// TIA Portal V17 export
// export: Created 2025-03-05T08:00:04.2235864Z, ExportSetting WithDefaults, DisplayName Totally Integrated Automation Portal, DisplayVersion V17 Update 8, DisplayName TIA Portal Openness, DisplayVersion V17 Update 8, DisplayName TIA Portal Version Control Interface, DisplayVersion V17, DisplayName SINAMICS Startdrive Advanced, DisplayVersion V17 SP2, DisplayName SINAMICS Startdrive G110M, G120, G120C, G120D, G120P, G115D, DisplayVersion V17 SP2, DisplayName SINAMICS Startdrive G130, G150, S120, S150, SINAMICS MV, S210, DisplayVersion V17 SP2, DisplayName STEP 7 Professional, DisplayVersion V17 Update 8, DisplayName SINUMERIK ONE STEP 7 Toolbox, DisplayVersion V17 Update 12, DisplayName SINUMERIK 840D sl STEP 7 Toolbox, DisplayVersion V17 Update 12, DisplayName STEP 7 Safety, DisplayVersion V17 Update 6, DisplayName WinCC Advanced, DisplayVersion V17 Update 8
FUNCTION "FC2037_GANTRY_ROBOT_TEST_CYCLE" : Void   // FC2037, LAD
{ S7_Optimized_Access := 'FALSE' }
AUTHOR : ETXETAR
VERSION : 1.0
// stored: AutoNumber false, IsIECCheckEnabled false, SetENOAutomatically false, UDAEnableTagReadback false
   VAR CONSTANT
      FC_NUMBER : DInt := 2037;
   END_VAR
   VAR_TEMP   // added for the SCL form of the ladder/FBD networks
      _w1 : Bool;
      _w2 : Bool;
   END_VAR
BEGIN

REGION Network 1: CHANGE CYCLE GENERAL CONDITIONS
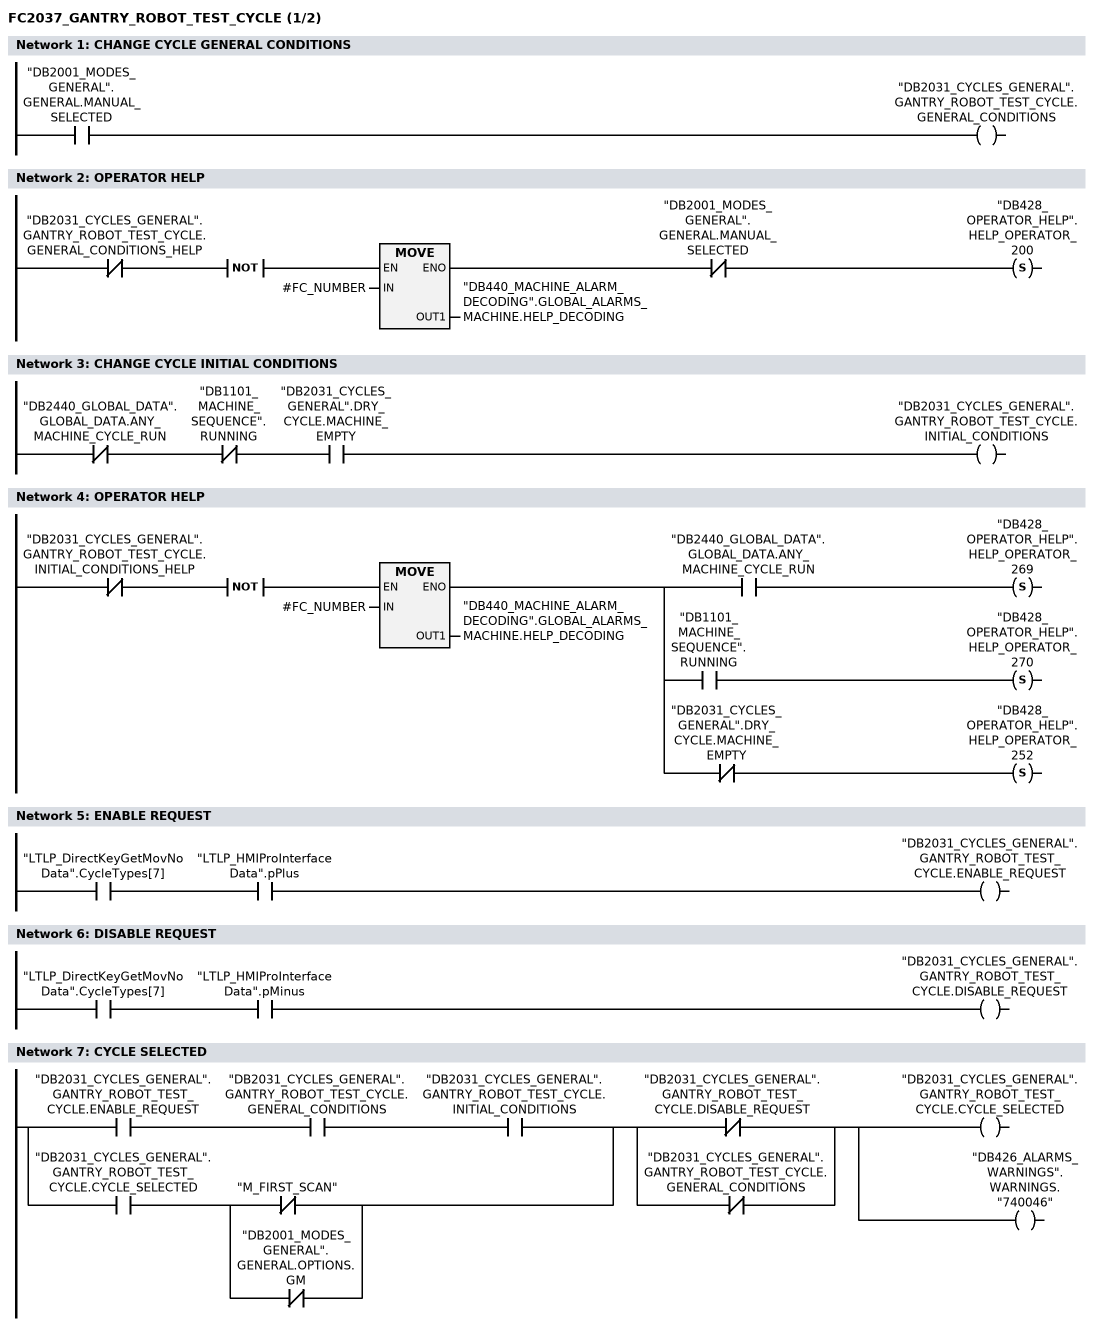
   RUNG wire#powerrail
      Contact( "DB2001_MODES_GENERAL".GENERAL.MANUAL_SELECTED )
      Coil( "DB2031_CYCLES_GENERAL".GANTRY_ROBOT_TEST_CYCLE.GENERAL_CONDITIONS )
   END_RUNG
   // the same network as SCL:
   "DB2031_CYCLES_GENERAL".GANTRY_ROBOT_TEST_CYCLE.GENERAL_CONDITIONS := "DB2001_MODES_GENERAL".GENERAL.MANUAL_SELECTED;
END_REGION

REGION Network 2: OPERATOR HELP
   RUNG wire#powerrail
      I_Contact( "DB2031_CYCLES_GENERAL".GANTRY_ROBOT_TEST_CYCLE.GENERAL_CONDITIONS_HELP )
      Not()
      { S7_GenerateENO := "TRUE" } Move(in := #FC_NUMBER, out1 => "DB440_MACHINE_ALARM_DECODING".GLOBAL_ALARMS_MACHINE.HELP_DECODING)
      I_Contact( "DB2001_MODES_GENERAL".GENERAL.MANUAL_SELECTED )
      S_Coil( "DB428_OPERATOR_HELP".HELP_OPERATOR_200 )
   END_RUNG
   // the same network as SCL:
   // ENO of a box is taken as its EN; it also drops when the box reports an error
   #_w1 := NOT (NOT "DB2031_CYCLES_GENERAL".GANTRY_ROBOT_TEST_CYCLE.GENERAL_CONDITIONS_HELP);
   IF #_w1 THEN "DB440_MACHINE_ALARM_DECODING".GLOBAL_ALARMS_MACHINE.HELP_DECODING := #FC_NUMBER; END_IF;
   IF #_w1 AND NOT "DB2001_MODES_GENERAL".GENERAL.MANUAL_SELECTED THEN
       "DB428_OPERATOR_HELP".HELP_OPERATOR_200 := TRUE;
   END_IF;
END_REGION

REGION Network 3: CHANGE CYCLE INITIAL CONDITIONS
   RUNG wire#powerrail
      I_Contact( "DB2440_GLOBAL_DATA".GLOBAL_DATA.ANY_MACHINE_CYCLE_RUN )
      I_Contact( "DB1101_MACHINE_SEQUENCE".RUNNING )
      Contact( "DB2031_CYCLES_GENERAL".DRY_CYCLE.MACHINE_EMPTY )
      Coil( "DB2031_CYCLES_GENERAL".GANTRY_ROBOT_TEST_CYCLE.INITIAL_CONDITIONS )
   END_RUNG
   // the same network as SCL:
   "DB2031_CYCLES_GENERAL".GANTRY_ROBOT_TEST_CYCLE.INITIAL_CONDITIONS := NOT "DB2440_GLOBAL_DATA".GLOBAL_DATA.ANY_MACHINE_CYCLE_RUN AND NOT "DB1101_MACHINE_SEQUENCE".RUNNING AND "DB2031_CYCLES_GENERAL".DRY_CYCLE.MACHINE_EMPTY;
END_REGION

REGION Network 4: OPERATOR HELP
   RUNG wire#powerrail
      I_Contact( "DB2031_CYCLES_GENERAL".GANTRY_ROBOT_TEST_CYCLE.INITIAL_CONDITIONS_HELP )
      Not()
      { S7_GenerateENO := "TRUE" } Move(in := #FC_NUMBER, out1 => "DB440_MACHINE_ALARM_DECODING".GLOBAL_ALARMS_MACHINE.HELP_DECODING)
      wire#w1
      Contact( "DB2440_GLOBAL_DATA".GLOBAL_DATA.ANY_MACHINE_CYCLE_RUN )
      S_Coil( "DB428_OPERATOR_HELP".HELP_OPERATOR_269 )
   END_RUNG
   RUNG wire#w1
      Contact( "DB1101_MACHINE_SEQUENCE".RUNNING )
      S_Coil( "DB428_OPERATOR_HELP".HELP_OPERATOR_270 )
   END_RUNG
   RUNG wire#w1
      I_Contact( "DB2031_CYCLES_GENERAL".DRY_CYCLE.MACHINE_EMPTY )
      S_Coil( "DB428_OPERATOR_HELP".HELP_OPERATOR_252 )
   END_RUNG
   // the same network as SCL:
   // ENO of a box is taken as its EN; it also drops when the box reports an error
   #_w1 := NOT (NOT "DB2031_CYCLES_GENERAL".GANTRY_ROBOT_TEST_CYCLE.INITIAL_CONDITIONS_HELP);
   IF #_w1 THEN "DB440_MACHINE_ALARM_DECODING".GLOBAL_ALARMS_MACHINE.HELP_DECODING := #FC_NUMBER; END_IF;
   IF #_w1 AND "DB2440_GLOBAL_DATA".GLOBAL_DATA.ANY_MACHINE_CYCLE_RUN THEN
       "DB428_OPERATOR_HELP".HELP_OPERATOR_269 := TRUE;
   END_IF;
   IF #_w1 AND "DB1101_MACHINE_SEQUENCE".RUNNING THEN
       "DB428_OPERATOR_HELP".HELP_OPERATOR_270 := TRUE;
   END_IF;
   IF #_w1 AND NOT "DB2031_CYCLES_GENERAL".DRY_CYCLE.MACHINE_EMPTY THEN
       "DB428_OPERATOR_HELP".HELP_OPERATOR_252 := TRUE;
   END_IF;
END_REGION

REGION Network 5: ENABLE REQUEST
   RUNG wire#powerrail
      Contact( "LTLP_DirectKeyGetMovNoData".CycleTypes[7] )
      Contact( "LTLP_HMIProInterfaceData".pPlus )
      Coil( "DB2031_CYCLES_GENERAL".GANTRY_ROBOT_TEST_CYCLE.ENABLE_REQUEST )
   END_RUNG
   // the same network as SCL:
   "DB2031_CYCLES_GENERAL".GANTRY_ROBOT_TEST_CYCLE.ENABLE_REQUEST := "LTLP_DirectKeyGetMovNoData".CycleTypes[7] AND "LTLP_HMIProInterfaceData".pPlus;
END_REGION

REGION Network 6: DISABLE REQUEST
   RUNG wire#powerrail
      Contact( "LTLP_DirectKeyGetMovNoData".CycleTypes[7] )
      Contact( "LTLP_HMIProInterfaceData".pMinus )
      Coil( "DB2031_CYCLES_GENERAL".GANTRY_ROBOT_TEST_CYCLE.DISABLE_REQUEST )
   END_RUNG
   // the same network as SCL:
   "DB2031_CYCLES_GENERAL".GANTRY_ROBOT_TEST_CYCLE.DISABLE_REQUEST := "LTLP_DirectKeyGetMovNoData".CycleTypes[7] AND "LTLP_HMIProInterfaceData".pMinus;
END_REGION

REGION Network 7: CYCLE SELECTED
   RUNG wire#powerrail
      Contact( "DB2031_CYCLES_GENERAL".GANTRY_ROBOT_TEST_CYCLE.ENABLE_REQUEST )
      Contact( "DB2031_CYCLES_GENERAL".GANTRY_ROBOT_TEST_CYCLE.GENERAL_CONDITIONS )
      Contact( "DB2031_CYCLES_GENERAL".GANTRY_ROBOT_TEST_CYCLE.INITIAL_CONDITIONS )
      wire#w1
      I_Contact( "DB2031_CYCLES_GENERAL".GANTRY_ROBOT_TEST_CYCLE.DISABLE_REQUEST )
      wire#w3
      Coil( "DB2031_CYCLES_GENERAL".GANTRY_ROBOT_TEST_CYCLE.CYCLE_SELECTED )
   END_RUNG
   RUNG wire#powerrail
      Contact( "DB2031_CYCLES_GENERAL".GANTRY_ROBOT_TEST_CYCLE.CYCLE_SELECTED )
      wire#w2
      I_Contact( "M_FIRST_SCAN" )
   END_RUNG wire#w1
   RUNG wire#w2
      I_Contact( "DB2001_MODES_GENERAL".GENERAL.OPTIONS.GM )
   END_RUNG wire#w1
   RUNG wire#w1
      I_Contact( "DB2031_CYCLES_GENERAL".GANTRY_ROBOT_TEST_CYCLE.GENERAL_CONDITIONS )
   END_RUNG wire#w3
   RUNG wire#w3
      Coil( "DB426_ALARMS_WARNINGS".WARNINGS."740046" )
   END_RUNG
   // the same network as SCL:
   "DB2031_CYCLES_GENERAL".GANTRY_ROBOT_TEST_CYCLE.CYCLE_SELECTED := (("DB2031_CYCLES_GENERAL".GANTRY_ROBOT_TEST_CYCLE.ENABLE_REQUEST AND "DB2031_CYCLES_GENERAL".GANTRY_ROBOT_TEST_CYCLE.GENERAL_CONDITIONS AND "DB2031_CYCLES_GENERAL".GANTRY_ROBOT_TEST_CYCLE.INITIAL_CONDITIONS) OR ("DB2031_CYCLES_GENERAL".GANTRY_ROBOT_TEST_CYCLE.CYCLE_SELECTED AND (NOT "M_FIRST_SCAN" OR NOT "DB2001_MODES_GENERAL".GENERAL.OPTIONS.GM))) AND (NOT "DB2031_CYCLES_GENERAL".GANTRY_ROBOT_TEST_CYCLE.DISABLE_REQUEST OR NOT "DB2031_CYCLES_GENERAL".GANTRY_ROBOT_TEST_CYCLE.GENERAL_CONDITIONS);
   "DB426_ALARMS_WARNINGS".WARNINGS."740046" := "DB2031_CYCLES_GENERAL".GANTRY_ROBOT_TEST_CYCLE.CYCLE_SELECTED;
END_REGION

REGION Network 8: WARNINGS
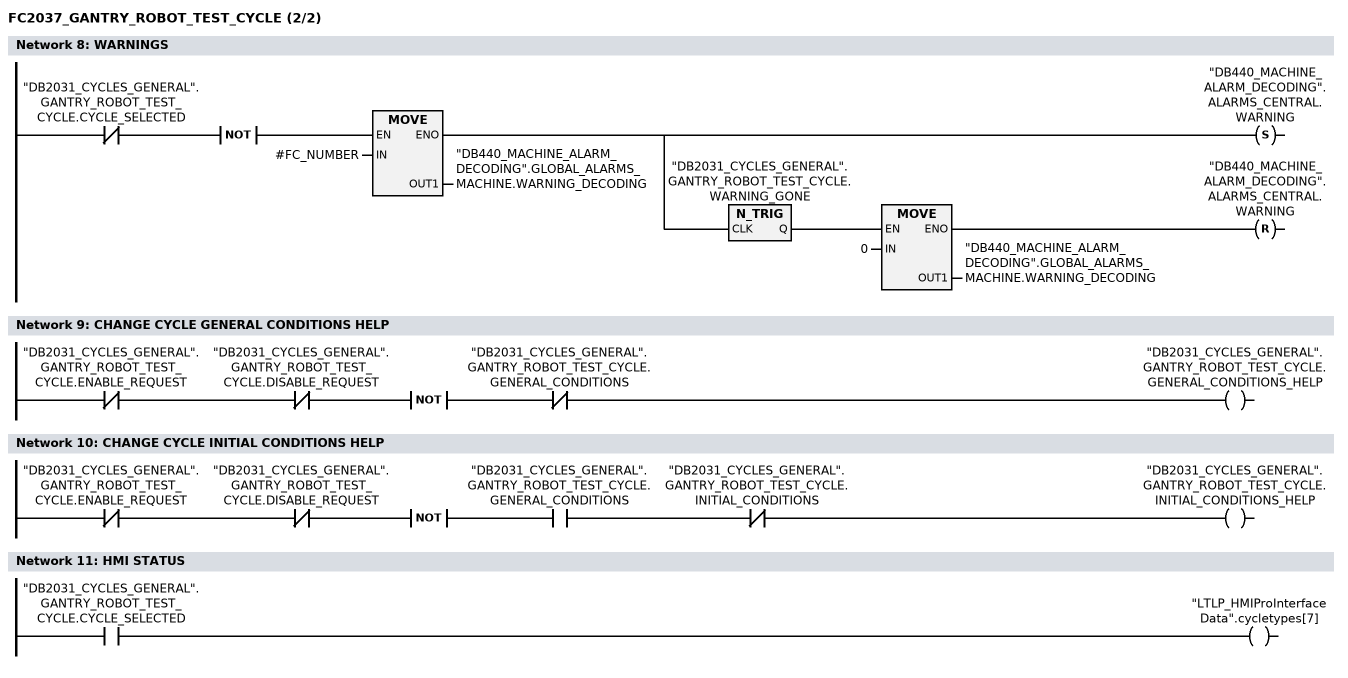
   RUNG wire#powerrail
      I_Contact( "DB2031_CYCLES_GENERAL".GANTRY_ROBOT_TEST_CYCLE.CYCLE_SELECTED )
      Not()
      Move(in := #FC_NUMBER, out1 => "DB440_MACHINE_ALARM_DECODING".GLOBAL_ALARMS_MACHINE.WARNING_DECODING)
      wire#w1
      S_Coil( "DB440_MACHINE_ALARM_DECODING".ALARMS_CENTRAL.WARNING )
   END_RUNG
   RUNG wire#w1
      N_Trig( "DB2031_CYCLES_GENERAL".GANTRY_ROBOT_TEST_CYCLE.WARNING_GONE )
      Move(in := 0, out1 => "DB440_MACHINE_ALARM_DECODING".GLOBAL_ALARMS_MACHINE.WARNING_DECODING)
      R_Coil( "DB440_MACHINE_ALARM_DECODING".ALARMS_CENTRAL.WARNING )
   END_RUNG
   // the same network as SCL:
   #_w1 := NOT (NOT "DB2031_CYCLES_GENERAL".GANTRY_ROBOT_TEST_CYCLE.CYCLE_SELECTED);
   IF #_w1 THEN
       "DB440_MACHINE_ALARM_DECODING".GLOBAL_ALARMS_MACHINE.WARNING_DECODING := #FC_NUMBER;
       "DB440_MACHINE_ALARM_DECODING".ALARMS_CENTRAL.WARNING := TRUE;
   END_IF;
   #_w2 := NOT #_w1 AND "DB2031_CYCLES_GENERAL".GANTRY_ROBOT_TEST_CYCLE.WARNING_GONE;   // falling edge
   "DB2031_CYCLES_GENERAL".GANTRY_ROBOT_TEST_CYCLE.WARNING_GONE := #_w1;
   IF #_w2 THEN
       "DB440_MACHINE_ALARM_DECODING".GLOBAL_ALARMS_MACHINE.WARNING_DECODING := 0;
       "DB440_MACHINE_ALARM_DECODING".ALARMS_CENTRAL.WARNING := FALSE;
   END_IF;
END_REGION

REGION Network 9: CHANGE CYCLE GENERAL CONDITIONS HELP
   RUNG wire#powerrail
      I_Contact( "DB2031_CYCLES_GENERAL".GANTRY_ROBOT_TEST_CYCLE.ENABLE_REQUEST )
      I_Contact( "DB2031_CYCLES_GENERAL".GANTRY_ROBOT_TEST_CYCLE.DISABLE_REQUEST )
      Not()
      I_Contact( "DB2031_CYCLES_GENERAL".GANTRY_ROBOT_TEST_CYCLE.GENERAL_CONDITIONS )
      Coil( "DB2031_CYCLES_GENERAL".GANTRY_ROBOT_TEST_CYCLE.GENERAL_CONDITIONS_HELP )
   END_RUNG
   // the same network as SCL:
   "DB2031_CYCLES_GENERAL".GANTRY_ROBOT_TEST_CYCLE.GENERAL_CONDITIONS_HELP := NOT (NOT "DB2031_CYCLES_GENERAL".GANTRY_ROBOT_TEST_CYCLE.ENABLE_REQUEST AND NOT "DB2031_CYCLES_GENERAL".GANTRY_ROBOT_TEST_CYCLE.DISABLE_REQUEST) AND NOT "DB2031_CYCLES_GENERAL".GANTRY_ROBOT_TEST_CYCLE.GENERAL_CONDITIONS;
END_REGION

REGION Network 10: CHANGE CYCLE INITIAL CONDITIONS HELP
   RUNG wire#powerrail
      I_Contact( "DB2031_CYCLES_GENERAL".GANTRY_ROBOT_TEST_CYCLE.ENABLE_REQUEST )
      I_Contact( "DB2031_CYCLES_GENERAL".GANTRY_ROBOT_TEST_CYCLE.DISABLE_REQUEST )
      Not()
      Contact( "DB2031_CYCLES_GENERAL".GANTRY_ROBOT_TEST_CYCLE.GENERAL_CONDITIONS )
      I_Contact( "DB2031_CYCLES_GENERAL".GANTRY_ROBOT_TEST_CYCLE.INITIAL_CONDITIONS )
      Coil( "DB2031_CYCLES_GENERAL".GANTRY_ROBOT_TEST_CYCLE.INITIAL_CONDITIONS_HELP )
   END_RUNG
   // the same network as SCL:
   "DB2031_CYCLES_GENERAL".GANTRY_ROBOT_TEST_CYCLE.INITIAL_CONDITIONS_HELP := NOT (NOT "DB2031_CYCLES_GENERAL".GANTRY_ROBOT_TEST_CYCLE.ENABLE_REQUEST AND NOT "DB2031_CYCLES_GENERAL".GANTRY_ROBOT_TEST_CYCLE.DISABLE_REQUEST) AND "DB2031_CYCLES_GENERAL".GANTRY_ROBOT_TEST_CYCLE.GENERAL_CONDITIONS AND NOT "DB2031_CYCLES_GENERAL".GANTRY_ROBOT_TEST_CYCLE.INITIAL_CONDITIONS;
END_REGION

REGION Network 11: HMI STATUS
   RUNG wire#powerrail
      Contact( "DB2031_CYCLES_GENERAL".GANTRY_ROBOT_TEST_CYCLE.CYCLE_SELECTED )
      Coil( "LTLP_HMIProInterfaceData".cycletypes[7] )
   END_RUNG
   // the same network as SCL:
   "LTLP_HMIProInterfaceData".cycletypes[7] := "DB2031_CYCLES_GENERAL".GANTRY_ROBOT_TEST_CYCLE.CYCLE_SELECTED;
END_REGION
END_FUNCTION
